Fanuc KAREL source: kt00517.KL

-- PROVISIONAL review KL for V940-1; original PC SHA256 158587b22a86ccacb2746c0b0935127e532e9f056c4ddf1be0119101b4dd9d36
-- Incomplete behavior may be omitted. Consult companion uncertainty JSON. Do not deploy.
PROGRAM KT00517
%NOLOCKGROUP
-- UNRESOLVED_DECL P1 type=000106
-- UNRESOLVED_DECL P2 type=000101
-- UNRESOLVED_DECL OUT type=000199
BEGIN
  -- V9_ZERO_TABLE_METADATA_HINT layout=0001; no indexed target words; source/name/runtime held
  -- UNRESOLVED_PC offsets 5-20; opcodes 2E,22,32,35
  -- UNRESOLVED_PC offsets 25-59; opcodes 49,7E,49,60,7E,4A
  -- UNRESOLVED_PC offsets 64-68; opcodes 7F
END KT00517
